FUNCTION F_LTIME_ARG : ST_Arg
VAR_INPUT
	tInput : LTIME;
END_VAR
VAR
	stArg : ST_Arg;
	sysVar_Info : __SYSTEM.VAR_INFO;
END_VAR

sysVar_Info 	:= __VARINFO(tInput);
stArg.TypeClass := sysVar_Info.TypeClass;
stArg.pValue 	:= 0;
stArg.diSize 	:= SIZEOF(tInput);
stArg.sValue 	:= TO_STRING(tInput); 
F_LTIME_ARG := stArg;

END_FUNCTION

(* stored: Version 1.1.0.1, ProductVersion 3.1.4024.4
   POU F_LTIME_ARG: Id {37de3b44-1334-460a-b0f4-1886875f4d2d}, SpecialFunc None *)
